ABB RobotStudio station: EstaciónDeSoldadura_20200720-170536.rsstn

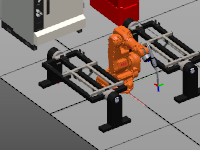
Station EstaciónDeSoldadura (saved by RobotStudio 7.0.8746.631)
Controller IRB_140_6kg_0.81m
  mechanical unit ROB_1: IRB140_6_81_C_03, 6 joints, base frame (0, 0, 0) mm
Layout (positions relative to the parent item):
  - IRB140_6_81_C_03 [mechanism, from Robots\IRB140_6_81_C_G_03.rslib] at (0, 0, 0) mm; joint values [0, 0, 0, 0, 0.5236, 0] (rad or m)
  - AW_Gun_PSF_25 [mechanism, from Tools\AW_Gun_PSF_25.rslib] at (506.29, 0, 679.5) mm, rotated rx 180 ry 60 rz 180 deg
  - IRC5_Singel-Cabinet [part, from Equipment\IRC5_Singel-Cabinet.rslib] at (-1350, 0, 100) mm, rotated rx 90 ry 0 rz 90 deg
  - Fronius_TPS4000_rev0 [part, from Equipment\Fronius_TPS4000.rslib] at (-1350, 900, 0) mm, rotated rx 0 ry 0 rz -90 deg
  - FlexPendant [part, from Equipment\FlexPendant.rslib] at (-1350, 0, 1100) mm, rotated rx 0 ry 0 rz 90 deg
  - Mesa [mechanism] at (-540, -540, 0) mm; joint values [0] (rad or m)
      links: L1, L2, L3
  - Mesa_2 [mechanism] at (-540, 540, 0) mm; joint values [0] (rad or m)
      links: L1, L2, L3
Attachment: AW_Gun_PSF_25 is attached to IRB140_6_81_C_03 / Link6
Targets, tools, work objects and paths stored in the station, written as RAPID:
! task T_ROB1
MODULE CalibData
  PERS tooldata AW_Gun:=[TRUE,[[119.5,0,352],[0.890213743,0,0.455543074,0]],[1,[0,0,100],[1,0,0,0],0,0,0]];
ENDMODULE

